// TIA Portal V18 export
TYPE "MEStoPLC_PrintExchange_ext"
// stored: IsFailsafeCompliant false
   STRUCT
      Load_PrintReqOK : Bool;   // 打标请求数据下发OK
      Load_PrintReqNG : Bool;   // 打标请求数据下发NG
      Load_PrintReqDone : Bool;   // 打标请求数据下发结束，PLC复位 PLC.Load_PrintReq
      Load_DataMatrixCheckOK : Bool;   // 二维码查询结果OK
      Load_DataMatrixCheckNG : Bool;   // 二维码查询结果NG
      Load_DataMatrixCheckDone : Bool;   // 二维码查询结束
      Spare : Bool;   // Spare
      Spare_1 : Bool;   // Spare
      SpareByte : Byte;   // SpareByte
      SpareByte_1 : Byte;   // SpareByte
   END_STRUCT;
END_TYPE
